PROGRAM V0_8
VAR
	fbOn : R_TRIG;
	fbOff : R_TRIG;
	
	bOnTrigger : BOOL;
	bOffTrigger : BOOL;
END_VAR

(*
	Teleruptorschakeling
	
	Programmeer de teleruptorschakeling in Structured Tekst. Zorg ook hier dat het mogelijk is om te bedienen met meerdere drukknoppen. Je zal merken dat dit een veel eenvoudiger programma zal zijn dan in LADDER. 

	Voor de flank-detectie heb je een Function Block (FB) nodig. Met een rechtermuisklik in het programmeervenster (niet het declareer venster) kan de 'input assisant' openen en selecteer vervolgens > Function Blocks > Tc2_Standard > trigger > R_TRIG
*)

fbOn(CLK := GVL.bButton_1 OR GVL.bButton_2, Q => bOnTrigger);
fbOff(CLK := GVL.bButton_3 OR GVL.bButton_4, Q => bOffTrigger);

GVL.bLamp_1 S= bOnTrigger;
GVL.bLamp_1 R= bOffTrigger;

END_PROGRAM

(* stored: Version 1.1.0.1, ProductVersion 3.1.4024.12
   POU V0_8: Id {a2eb5d76-f3b7-4ebc-a5db-20c9f3d4c026}, SpecialFunc None *)
